# EPICS substitutions: ssaApp/Db/ssa_sys0_common.substitutions
# Common controls for sys0 (all SC linac) SSAs.
# Required macros:
#   OUT: PV attribute

file "ssaCommonControls_sys0.template" {
pattern
{     OUT,      ZNAM,        ONAM, DLY}
{PowerOff, "Standby", "Power Off", 0.1}
}
